(* PLC project Generated.project, CODESYS CODESYS V3.5 SP19 Patch 1 *)
(* stored: creationDateTime 2026-09-06T13:00:42.542779, modificationDateTime 2026-09-06T13:00:42.542779 *)

(* ═══════════════════════════════════════════════════════════════ 🎮 ST_JoystickCmd — Commandes IHM pour le Joystick ═══════════════════════════════════════════════════════════════ *)
TYPE ST_JoystickCmd : STRUCT
  Calibrate : BOOL;  (* 🎯 Demande de recalage au neutre (front) *)
END_STRUCT;
END_TYPE
